{attribute addProperty BoxType "KL9900-0059"}
{attribute addProperty Id "Channel_1Channel_40E5A7A500"}
{attribute addProperty CRC "2836401290"}
{attribute addProperty SizeInBites "0"}
{attribute addProperty SizeInBytes "0"}
TYPE KL_A9100C8A :
STRUCT
	{attribute addProperty Name "Channel_1"}
	Channel_1 : Channel_40E5A7A5;
END_STRUCT
END_TYPE

(* stored: Version 1.2.0.0, ProductVersion 3.1.4024.9
   DUT KL_A9100C8A: Id {2a387fd3-4e37-4f95-b62a-d5556a2aad97} *)
